(* CODESYS project Tc Motion Control.library
   Version: 0.1.0.0
   Title: Motion
   Author: Adam Garner
   Placeholder: Motion
   Company: Ljmu

Project tree, tasks and I/O mapping:
  libraries: Tc2_MC2, * (Beckhoff Automation GmbH); Tc2_MC2_Drive, * (Beckhoff Automation GmbH); Tc2_Standard, * (Beckhoff Automation GmbH); Tc2_System, * (Beckhoff Automation GmbH); Tc2_Utilities, * (Beckhoff Automation GmbH); Tc3_EventLogger, * (Beckhoff Automation GmbH); Tc3_JsonXml, * (Beckhoff Automation GmbH); Tc3_Module, * (Beckhoff Automation GmbH)
  DUTs/
    data type e_IDXBrakeState
    data type e_IDXError
    data type e_MCState
    data type e_MotorReadState
    data type ST_IDXError
    data type ST_IDXErrorCode
    data type ST_MCState
  GVLs/
  POUs/
    function block FB_IDXError [ST]: FB_init, GetErrorStructure, IsError, ResetError
    function block FB_IDXReadErrorCode [ST]: ParseErrorCode
    function block FB_IDXReadErrorRegister [ST]: ParseErrorRegister
    function block FB_IDXResetError [ST]: FB_init
    function block FB_Motion [ST]: Enable, Estop, FB_init, GetAxisRef, GetCurrentPosition, GetStatus, Home, MoveTo, Reset
    function block FB_MotionEventSender [ST]: COEError, EnableMotor, Homing, MotorError, MotorReset, MoveTo, NCError, NCReset
    function block FB_MotorBrake [ST]: Brake, BrakeStatus, EnableMotor, FB_init, UnitTestInputs
    function block FB_ReadErrorStringFromESI [ST]: FB_init, GetErrorString, StringToUint
    program MAIN [ST]
  VISUs/
*)

// DUTs/e_IDXBrakeState
{attribute 'qualified_only'}
{attribute 'strict'}
TYPE e_IDXBrakeState :
(
	Unpowered := 0,// no air in system brake on 
	Disengaging := 1, // Brake coming off 
	Disengaged :=2,// held off with compressed air
	Engaging	:=3, // brake coming online under command
	Engaged	:= 4,// brake on air in system 
	SafetyOverriden := 5, // safety override on brake on 
	SafetyActivating := 6, // safety override on brake Activing
	Unknown := 7,
	Error := 8
);
END_TYPE

// DUTs/e_IDXError
{attribute 'qualified_only'}
{attribute 'strict'}
TYPE e_IDXError :
(
	Generic_Error := 0,
	Current_Error :=1,
	Voltage_Error:=2,
	Temperature_Error:=3,
	Communication_Error := 4,
	Device_Profile_Specific := 5,
	Reserved := 6,
	Motion_Error :=7
);
END_TYPE

// DUTs/e_MCState
{attribute 'qualified_only'}
{attribute 'strict'}
TYPE e_MCState :
(
	Busy,
	Done,
	Error,
	CommandAborted,
	Active,
	Idle
);
END_TYPE

// DUTs/e_MotorReadState
// -27 as is qualified only shouldnt be flagged anyway
{attribute 'strict'}
{attribute 'qualified_only'}
TYPE e_MotorReadState :
(
Idle,
ReadingErrorArray,
{attribute 'analysis' := '-27'}
Parse,
EraseErrorArray,
Waiting,
Error,
CountingErrors,
ReadNextError

);
END_TYPE

// DUTs/ST_IDXError
TYPE ST_IDXError :
STRUCT
	GenericError:BOOL;
	CurrentError : BOOL;
	VoltageError:BOOL;
	TemperatureError:BOOL;
	Communication_Error :BOOL;
	DeviceProfileSpecific :BOOL;
	Reserved :BOOL;
	MotionError :BOOL;
	ErrorCodeArr:ARRAY [0..4] OF ST_IDXErrorCode;


END_STRUCT
END_TYPE

// DUTs/ST_IDXErrorCode
TYPE ST_IDXErrorCode :
STRUCT
	ErrorCode: UINT;
	ErrorString:STRING;
	TimeCode:DT;
END_STRUCT
END_TYPE

// DUTs/ST_MCState
TYPE ST_MCState :
STRUCT
	MCState : e_MCState;
	Done:BOOL;
	CommandAborted:BOOL;
	Status :BOOL;
	Active :BOOL;
	Busy:BOOL;
	Error:BOOL;
	ErrorID:UDINT;
	
END_STRUCT
END_TYPE

// POUs/FB_IDXError
FUNCTION_BLOCK FB_IDXError
// www.maxongroup.com/medias/sys_master/root/8837359632414/IDX-Firmware-Specification-En.pdf 	
VAR
	AxisName 				:STRING;
	ExecuteRead 			: BOOL; 
	MappedErrorCode AT%I* 	: UINT;
	stIDXError 				: ST_IDXError;
	
	fbIDXErrorEventSender 	: FB_MotionEventSender;
	MotorErrorEventSent		: BOOL;


	fbIdxReadErrorCode 		: FB_IDXReadErrorCode;
	NumOfErrorCodes			: USINT;
	ErrorCodeReadError 		: BOOL;
	ErrorCodeAdsErrorCode	: UINT;
	ErrorCodeReadBusy		: BOOL;
	
	fbIDXReadErrorRegister	: FB_IDXReadErrorRegister;
	ErrorRegisterReadError 	: BOOL;
	ErrorRegisterReadBusy	: BOOL;
	ErrorRegisterAdsErrorCode: UINT;
	
	fbReadErrorStringFromESI: FB_ReadErrorStringFromESI(FileNameIn := 'C:\ProgramData\Beckhoff\TwinCAT\3.1\Repository\Beckhoff Automation GmbH\maxon_motor_IDX_0170h_6650h_0000h_0000h_ESI.xml');
	ErrorStringReadReady 	: BOOL;
	ErrorStringReadBusy 	: BOOL;
	ErrorStringReadError 	: BOOL;
	ErrorStringFound 		: BOOL;
	
	CoeErrorCodeMessageSent : BOOL;
	CoeErrorregisterMessageSent : BOOL;
	
	

	

END_VAR

VAR_INPUT
	Axis 					: AXIS_REF;
END_VAR

VAR_OUTPUT
    Busy         			: BOOL;
    Error        			: BOOL;
END_VAR

VAR CONSTANT
	MaxIndex 				: USINT := 4;
END_VAR

VAR_TEMP
	TempErrorCode 			: UINT;
	TempErrorString 		: STRING;
	Index					: USINT;
END_VAR

// read error Reg 
// check for error messages availible 

IF NOT (MappedErrorCode=0) THEN
	ExecuteRead := TRUE; // motor in error state 
	
ELSE
	ExecuteRead:= FALSE;
END_IF

fbIdxReadErrorCode(
	Axis:= Axis,
	Execute:= ExecuteRead,
	NumOfErrors=> NumOfErrorCodes,
	stErrorInOut:=stIDXError,
	ReadError=>ErrorCodeReadError,
	AdsErrId=>ErrorCodeAdsErrorCode,
	ReadBusy => ErrorCodeReadBusy);

CoeErrorCodeMessageSent := fbIDXErrorEventSender.COEError(
	AxisName := AxisName,
	Error := ErrorCodeReadError,
	AdsErrId:= ErrorCodeAdsErrorCode,
	Description:= 'ErrorCodeRead');

fbIDXReadErrorRegister(
	Axis:= Axis, 
	Execute:= ExecuteRead, 
	stErrorRegisterInOut:=stIDXError , 
	ReadError=> ErrorRegisterReadError, 
	AdsErrId=> ErrorRegisterAdsErrorCode, 
	ReadBusy=> ErrorRegisterReadBusy );

CoeErrorregisterMessageSent:= fbIDXErrorEventSender.COEError(
	AxisName:= AxisName,
	Error := ErrorRegisterReadError,
	AdsErrId:= ErrorRegisterAdsErrorCode,
	Description:= 'ErrorCodeRegister');


fbReadErrorStringFromESI(
	ReadyFlag=>ErrorStringReadReady,
	Busy=>ErrorStringReadBusy,
	Error=>ErrorStringReadError);


IF (ErrorStringReadReady AND ExecuteRead ) THEN
	FOR Index:=0  TO MaxIndex BY 1 DO
		TempErrorCode:= stIDXError.ErrorCodeArr[Index].ErrorCode;
		IF NOT (TempErrorCode =0) THEN
			ErrorStringFound:= fbReadErrorStringFromESI.GetErrorString(ErrorCodeIn:= TempErrorCode,ErrorStringOut=>TempErrorString);
			stIDXError.ErrorCodeArr[Index].ErrorString:= TempErrorString;
		END_IF
	END_FOR
END_IF
	
MotorErrorEventSent:= fbIDXErrorEventSender.MotorError(stIDXError:=stIDXError,AxisName:= AxisName);

Busy := ErrorStringReadBusy OR ErrorRegisterReadBusy OR ErrorCodeReadBusy;
Error := ErrorStringReadError OR ErrorRegisterReadError OR ErrorCodeReadError;

METHOD FB_init : BOOL
VAR_INPUT
	bInitRetains : BOOL; // if TRUE, the retain variables are initialized (warm start / cold start)
	bInCopyCode : BOOL;  // if TRUE, the instance afterwards gets moved into the copy code (online change)
	AxisNameIn	:String;
END_VAR
AxisName := AxisNameIn;
END_METHOD

METHOD PUBLIC GetErrorStructure 
VAR_OUTPUT
	StIDXErrorOut : ST_IDXError;
END_VAR
StIDXErrorOut:= stIDXError;
END_METHOD

// returns true if motor is in error state 
METHOD IsError : BOOL
IsError := ExecuteRead;
END_METHOD

METHOD ResetError : BOOL
VAR_IN_OUT
	   		{attribute 'analysis' := '-27'}
	Execute			: BOOL;(*Function block execution is triggered by a rising edge at this input.*)
END_VAR

VAR_INST
	fbCoEWrite		: FB_CoEWrite;
    Data       		: UINT := 16#0080;
    ReadError          	: BOOL;
    AdsErrId       	: UINT;
    CANopenErrId   	: UINT;
END_VAR

VAR CONSTANT
	NetId          	: T_AmsNetID:= '';(*netID of PC with NC*)
   	Index          	: WORD:= 16#6040;(*CoE object index*)
   	SubIndex       	: BYTE:=16#0;(*CoE sub index*)
   	Timeout        	: TIME := DEFAULT_ADS_TIMEOUT;(*States the time before the function is cancelled.*)
  	CompleteAccess 	: BOOL:= FALSE;(*Function block reads the complete object with all sub index*)
END_VAR
IF __ISVALIDREF(Execute) THEN	
	fbCoEWrite(
    NetId          := NetId, 
    Index          := Index, 
    SubIndex       := SubIndex, 
    pSrcBuf        := ADR(Data), 
    BufLen         := USINT_TO_UDINT(SIZEOF(Data)), 
    Execute        := Execute, 
    Timeout        := Timeout, 
    CompleteAccess := CompleteAccess, 
    Axis := Axis
);

END_IF

IF (NOT fbCoEWrite.Busy) AND   __ISVALIDREF(Execute) THEN
    ReadError    := fbCoEWrite.Error;
	IF (NOT ReadError) AND Execute THEN
		ResetError:= TRUE; // reset successfully only shows for one cycle
	ELSE 
		ResetError:= FALSE;
	END_IF
	
    AdsErrId     := fbCoEWrite.AdsErrId;
    CANopenErrId :=fbCoEWrite.CANopenErrId;
    Execute      := FALSE;
	IF NOT ReadError THEN
		ResetError:= TRUE; // reset successfully
	END_IF
END_IF
END_METHOD

END_FUNCTION_BLOCK

// POUs/FB_MotionEventSender
{attribute 'analysis' := '-2'} // empty function block
// this fb is used to generate events via methods used in this libary 
FUNCTION_BLOCK INTERNAL FB_MotionEventSender
VAR
	fbTcMessage : FB_TcMessage;
END_VAR

// returns true for one cycle when event is generated 
// method is used for events in a Coe read/write 
METHOD INTERNAL COEError : BOOL

VAR_INPUT
    Error        	: BOOL; // from COE read/write 
    AdsErrId     	: UINT; // from COE read/write 
	Description		: STRING; // description of what the COE was doing eg MotorError Read or MotorReset Write is displayed in event
	AxisName		:STRING; // for display in event 
END_VAR
VAR_INST //previous cycle results
	LastError		:BOOL; 

END_VAR

VAR
	SendResult 			:HRESULT;

END_VAR
COEError := FALSE;
IF (NOT LastError) AND Error THEN // only enter is a current error is in place and the last cycle the error was 0 
	 {analysis -9,-46} // Unused  return values and possible use of none init interfaces 
	fbTcMessage.CreateEx(TC_EVENTS.MotionEvents.CoeError,0);
	fbTcMessage.ipArguments.Clear();
	fbTcMessage.ipArguments.AddString(AxisName);
	fbTcMessage.ipArguments.AddUInt(AdsErrId);
	fbTcMessage.ipArguments.AddString(Description);
	SendResult:= fbTcMessage.Send(0);
	{analysis 9,46}
	IF (SendResult=0) THEN
		COEError := TRUE;
	END_IF
END_IF
LastError:= Error;
END_METHOD

// method generates events when axis is enabled / disabled 
// returns true for one cycle when event is generated 
METHOD INTERNAL EnableMotor 		: BOOL
VAR_IN_OUT
	stAxisPowerState 	: ST_MCState; //structure from fb motion libary shows movement FB status 
END_VAR
VAR_INPUT
	AxisName 			:STRING; // displayed in event 
END_VAR
VAR_INST //previous cycle results
	stLastAxisPowerState :ST_MCState;
END_VAR
VAR
	SendResult 			: HRESULT;
	SendEvent 			: BOOL := FALSE;
END_VAR
EnableMotor := FALSE;

IF __ISVALIDREF(stAxisPowerState) THEN

	IF NOT (stLastAxisPowerState.MCState = stAxisPowerState.MCState) THEN // state has changed 
	 	{analysis -9,-46} // Unused  return values and possible use of none init interfaces 
		CASE(stAxisPowerState.MCState) OF
		
		e_MCState.Active:
			fbTcMessage.CreateEx(TC_EVENTS.MotionEvents.MotorEnabled,0);
			SendEvent:= TRUE;
		
		e_MCState.Error:
			fbTcMessage.CreateEx(TC_EVENTS.MotionEvents.MotorEnableError,0);
			SendEvent:= TRUE;
		
		e_MCState.Idle:
			fbTcMessage.CreateEx(TC_EVENTS.MotionEvents.MotorDisabled,0);
			SendEvent:= TRUE;
		ELSE
			SendEvent:= FALSE;
		END_CASE
	
		IF SendEvent THEN
			fbTcMessage.ipArguments.Clear();
			fbTcMessage.ipArguments.AddString(AxisName);
			SendResult:= fbTcMessage.Send(0);
			IF (SendResult=0) THEN
				EnableMotor := TRUE;
			END_IF
		END_IF
	END_IF

	stLastAxisPowerState := stAxisPowerState;
END_IF
END_METHOD

// returns true for one cycle when event is generated 
// creates events during homing
// returns true for one cycle when event is generated 
METHOD INTERNAL Homing : BOOL
VAR_IN_OUT
	stAxisHomeState : ST_MCState; //structure from fb motion libary shows movement FB status 
END_VAR
VAR_INPUT
	AxisName :STRING; // displayed in event 
 
END_VAR
VAR_INST //previous cycle results
	stLastAxisHomeState : ST_MCState;
END_VAR
VAR
	SendEvent : BOOL;
	SendResult : Hresult;
END_VAR
Homing := FALSE;

IF  __ISVALIDREF(stAxisHomeState) THEN
	
	IF  (NOT (stLastAxisHomeState.MCState = stAxisHomeState.MCState)) THEN
		CASE(stAxisHomeState.MCState) OF 
		{analysis -9,-46} // Unused  return values and possible use of none init interfaces 
		e_MCState.Done:
			fbTcMessage.CreateEx(TC_EVENTS.MotionEvents.HomeCompleted,0);
			fbTcMessage.ipArguments.Clear();
			fbTcMessage.ipArguments.AddString(AxisName);
			SendEvent := TRUE;
		
		e_MCState.Busy:
			fbTcMessage.CreateEx(TC_EVENTS.MotionEvents.HomeCommandReceived,0);
			fbTcMessage.ipArguments.Clear();
			fbTcMessage.ipArguments.AddString(AxisName);
			SendEvent := TRUE;
		
		e_MCState.Error:
			fbTcMessage.CreateEx(TC_EVENTS.MotionEvents.HomeError,0);
			fbTcMessage.ipArguments.Clear();
			fbTcMessage.ipArguments.AddString(AxisName);
			fbTcMessage.ipArguments.AddUDInt(stAxisHomeState.ErrorID);
			SendEvent := TRUE;
			
		
		e_MCState.CommandAborted:
			fbTcMessage.CreateEx(TC_EVENTS.MotionEvents.HomeAborted,0);
			fbTcMessage.ipArguments.Clear();
			fbTcMessage.ipArguments.AddString(AxisName);
			SendEvent := TRUE;
			
		e_MCState.Idle:
			SendEvent := FALSE;
		
		ELSE
			SendEvent := FALSE;
			
		
		END_CASE
		
			IF SendEvent THEN
				SendResult:= fbTcMessage.Send(0);
			
				IF (SendResult=0) THEN
					Homing := TRUE;
				END_IF
	
			END_IF
	END_IF
	
	stLastAxisHomeState:= stAxisHomeState;

END_IF
END_METHOD

// genereates events about a motor controllers errors it loops through the array of data errors in St_IDXError
// returns true for one cycle when event is generated 
METHOD INTERNAL MotorError :BOOL
VAR_IN_OUT
	stIDXError 	:ST_IDXError;
END_VAR
VAR_INPUT
	AxisName 	:STRING;  // displayed in event 
END_VAR
VAR_INST //previous cycle results
	stLastIDXError : ST_IDXError;
END_VAR
VAR
	Index :INT;
	ErrorCodeInHex :STRING[255];
	SendResult :HRESULT;
END_VAR
VAR CONSTANT
	MaxIndex :INT := 4 ; // upper limit of loop 
END_VAR
MotorError:= FALSE;
IF __ISVALIDREF(stIDXError) THEN
FOR Index := 0 TO MaxIndex BY 1 DO 
	IF NOT ( stIDXError.ErrorCodeArr[Index].ErrorCode =stLastIDXError.ErrorCodeArr[Index].ErrorCode) THEN
		{analysis -9,-46,-130}// Unused  return values possible use of none init interfaces ,  Implicit expanding conversion 
		fbTcMessage.CreateEx(TC_EVENTS.MotionEvents.MotorError,0);
		fbTcMessage.ipArguments.Clear();
		fbTcMessage.ipArguments.AddString(AxisName);
		ErrorCodeInHex := DWORD_TO_HEXSTR(stIDXError.ErrorCodeArr[Index].ErrorCode,4,FALSE); // error code as hex string 
		fbTcMessage.ipArguments.AddString(ErrorCodeInHex);
		fbTcMessage.ipArguments.AddString(stIDXError.ErrorCodeArr[Index].ErrorString);
		SendResult := fbTcMessage.Send(0);
		{analysis 9,46,130}
		IF (SendResult=0) THEN
			MotorError:= TRUE;
		END_IF
		stLastIDXError.ErrorCodeArr[Index]:= stIDXError.ErrorCodeArr[Index];
			
	END_IF
END_FOR
END_IF
END_METHOD

// events for resetting a motor controller 
// returns true for one cycle when event is generated 
METHOD INTERNAL MotorReset : BOOL
VAR_IN_OUT
	stAxisResetState : ST_MCState;
END_VAR
VAR_INPUT
	AxisName :STRING; // displayed in event
	ErrorCodeIn :UDINT;
END_VAR
VAR_INST//previous cycle results
	stLastAxisResetState : ST_MCState;
END_VAR
VAR
	SendEvent : BOOL;
	SendResult : Hresult;
END_VAR
MotorReset := FALSE;

IF  __ISVALIDREF(stAxisResetState) THEN
	
	IF  (NOT (stLastAxisResetState.MCState = stAxisResetState.MCState)) THEN
		CASE(stAxisResetState.MCState) OF 
		{analysis -9,-46} // Unused  return values and possible use of none init interfaces 
		e_MCState.Done:
			fbTcMessage.CreateEx(TC_EVENTS.MotionEvents.MotorResetCompleted,0);
			fbTcMessage.ipArguments.Clear();
			fbTcMessage.ipArguments.AddString(AxisName);
			SendEvent := TRUE;
		
		e_MCState.Busy:
			fbTcMessage.CreateEx(TC_EVENTS.MotionEvents.MotorResetReceived,0);
			fbTcMessage.ipArguments.Clear();
			fbTcMessage.ipArguments.AddString(AxisName);
			SendEvent := TRUE;
		
		e_MCState.Error:
			SendEvent := FALSE;
			
		e_MCState.Idle:
			SendEvent := FALSE;
		
		ELSE
			SendEvent := FALSE;
			
		
		END_CASE
		
			IF SendEvent THEN
				SendResult:= fbTcMessage.Send(0);
			
				IF (SendResult=0) THEN
					MotorReset := TRUE;
				END_IF
	
			END_IF
	END_IF
	
	stLastAxisResetState:= stAxisResetState;

END_IF
END_METHOD

// method used to generate events on movement commands 
// moveTo bool is true when a event has been sent 
METHOD MoveTo : BOOL
VAR_IN_OUT
	stAxisMoveState : ST_MCState;
END_VAR
VAR_INPUT
	AxisName :STRING;// displayed in event
	TargetPositionIn : LREAL;
	VelocityIn : LREAL;
END_VAR
VAR_INST//previous cycle results
	stLastAxisMoveState : ST_MCState;
END_VAR
VAR
	SendEvent : BOOL;
	SendResult : Hresult;
	
END_VAR
MoveTo:= FALSE;
	
IF __ISVALIDREF(stAxisMoveState) THEN
	
	IF  (NOT (stAxisMoveState.MCState = stLastAxisMoveState.MCState)) THEN
	
		CASE(stAxisMoveState.MCState) OF 
		{analysis -9,-46} // Unused  return values and possible use of none init interfaces 	
			e_MCState.Active:
			fbTcMessage.CreateEx(TC_EVENTS.MotionEvents.MotorMoveActive,0);
			fbTcMessage.ipArguments.Clear();
			fbTcMessage.ipArguments.AddString(AxisName);
			SendEvent := TRUE;
	
		e_MCState.Busy:
			fbTcMessage.CreateEx(TC_EVENTS.MotionEvents.MoveCommandReceived,0);
			fbTcMessage.ipArguments.Clear();
			fbTcMessage.ipArguments.AddString(AxisName);
			fbTcMessage.ipArguments.AddLReal(TargetPositionIn);
			fbTcMessage.ipArguments.AddLReal(VelocityIn);
			SendEvent := TRUE;
	
		e_MCState.Error:
			fbTcMessage.CreateEx(TC_EVENTS.MotionEvents.MotorMoveError,0);
			fbTcMessage.ipArguments.Clear();
			fbTcMessage.ipArguments.AddString(AxisName);
			fbTcMessage.ipArguments.AddUDInt(stAxisMoveState.ErrorID);
			SendEvent := TRUE;
	
		e_MCState.CommandAborted:
			fbTcMessage.CreateEx(TC_EVENTS.MotionEvents.MovementAborted,0);
			fbTcMessage.ipArguments.Clear();
			fbTcMessage.ipArguments.AddString(AxisName);
			SendEvent := TRUE;
	
		e_MCState.Done:
			fbTcMessage.CreateEx(TC_EVENTS.MotionEvents.MotorMoveFinshed,0);
			fbTcMessage.ipArguments.Clear();
			fbTcMessage.ipArguments.AddString(AxisName);
			fbTcMessage.ipArguments.AddLReal(TargetPositionIn);
			SendEvent := TRUE;
	
		e_MCState.Idle:
			SendEvent := FALSE;
	
	
		ELSE
			SendEvent := FALSE;
		
		END_CASE
		
		IF SendEvent THEN
			SendResult:= fbTcMessage.Send(0);
			
			IF (SendResult=0) THEN
				MoveTo := TRUE;
			END_IF
		
		END_IF
	
		stLastAxisMoveState := stAxisMoveState;
	
	END_IF

END_IF
END_METHOD

// method creates events for NC block Errors 
// returns true for one cycle when event is generated 
METHOD INTERNAL NCError : BOOL
VAR_IN_OUT
	stAxisStatus : ST_AxisStatus;
END_VAR
VAR_INPUT
	AxisName 	:STRING; // displayed in event
END_VAR
VAR_INST//previous cycle results
	stLastAxisErrorID :UDINT;
END_VAR
VAR
	SendResult :HRESULT;
END_VAR
NCError:= FALSE;
IF __ISVALIDREF(stAxisStatus) THEN

	IF NOT ( stAxisStatus.ErrorID = stLastAxisErrorID) THEN
		{analysis -9,-46,-130}// Unused  return values possible use of none init interfaces ,  Implicit expanding conversion 
		fbTcMessage.CreateEx(TC_EVENTS.MotionEvents.NCError,0);
		fbTcMessage.ipArguments.Clear();
		fbTcMessage.ipArguments.AddString(AxisName);
		fbTcMessage.ipArguments.AddUDInt(stAxisStatus.ErrorID);
		SendResult := fbTcMessage.Send(0);
		{analysis 9,46,130}
		IF (SendResult=0) THEN
			NCError:= TRUE;
		END_IF
		stLastAxisErrorID:= stAxisStatus.ErrorID;
			
	END_IF
END_IF
END_METHOD

// creates events during a NCreset 
// returns true for one cycle when event is generated 
METHOD INTERNAL NCReset : BOOL
VAR_IN_OUT
	stAxisResetState : ST_MCState;
	
END_VAR
VAR_INPUT
	AxisName :STRING;// displayed in event
	ErrorCodeIn :UDINT;
END_VAR
VAR_INST//previous cycle results
	stLastAxisResetState : ST_MCState;
END_VAR
VAR
	SendEvent : BOOL;
	SendResult : Hresult;
END_VAR
NCReset := FALSE;

IF  __ISVALIDREF(stAxisResetState) THEN
	
	IF  (NOT (stLastAxisResetState.MCState = stAxisResetState.MCState)) THEN
		CASE(stAxisResetState.MCState) OF 
		{analysis -9,-46} // Unused  return values and possible use of none init interfaces 
		e_MCState.Done:
			fbTcMessage.CreateEx(TC_EVENTS.MotionEvents.NCResetCompleted,0);
			fbTcMessage.ipArguments.Clear();
			fbTcMessage.ipArguments.AddString(AxisName);
			SendEvent := TRUE;
		
		e_MCState.Busy:
			fbTcMessage.CreateEx(TC_EVENTS.MotionEvents.NCResetReceived,0);
			fbTcMessage.ipArguments.Clear();
			fbTcMessage.ipArguments.AddString(AxisName);
			SendEvent := TRUE;
		
		e_MCState.Error:
			fbTcMessage.CreateEx(TC_EVENTS.MotionEvents.NCResetError,0);
			fbTcMessage.ipArguments.Clear();
			fbTcMessage.ipArguments.AddString(AxisName);
			fbTcMessage.ipArguments.AddUDInt(ErrorCodeIn);
			SendEvent := TRUE;
			
		e_MCState.Idle:
			SendEvent := FALSE;
		
		ELSE
			SendEvent := FALSE;
			
		
		END_CASE
		
			IF SendEvent THEN
				SendResult:= fbTcMessage.Send(0);
			
				IF (SendResult=0) THEN
					NCReset := TRUE;
				END_IF
	
			END_IF
	END_IF
	
	stLastAxisResetState:= stAxisResetState;

END_IF
END_METHOD

END_FUNCTION_BLOCK

// POUs/FB_IDXReadErrorCode
// function to read the Diagnosis history odject of a IDX motor 
// this fb will read the errors in the error array looping between them with a 1s pause between reads
// if execute is false it resets the error array no none 
// www.maxongroup.com/medias/sys_master/root/8837359632414/IDX-Firmware-Specification-En.pdf
// definition of motor structure on 6.2.12 pg 71

FUNCTION_BLOCK FB_IDXReadErrorCode
VAR CONSTANT
	 NetId             : T_AmsNetID := ''; // assumes local machine 
    Index             : WORD := 16#10F3; // diagnosis history 
    Timeout           : TIME := T#5S;
    CompleteAccess    : BOOL := FALSE; // to read the whole index in one go instead of sunindexs
	NumberOfErrors :USINT := 5; // number of errors 
	MaxErrorIndex :USINT := 4; // max index so one below number of errors 
	MotorErrorSubindexStart :USINT := 6 ;
END_VAR
VAR_INPUT
	Axis :AXIS_REF;// used For Coe read 
		 {attribute 'analysis' := '-27'}
	Execute: BOOL;	
END_VAR
VAR_IN_OUT
	stErrorInOut : ST_IDXError;// a array for errors with code string and datetime 
END_VAR
VAR_OUTPUT
	NumOfErrors :USINT; // how man errors are present 
	ReadError :BOOL; // error reading motor 
	AdsErrId  : UINT; //holds Reading error codes 
	ReadBusy:BOOL;
END_VAR

VAR
	eMotorReadState : e_MotorReadState; // enum of fb  current state
	
	CoETimer : TON:= (PT:= T#1S); // timer 
	TimerStart:BOOL:= FALSE;
	TimerElapsed:BOOL;
	fbCoERead         : FB_CoERead; // fb to Coe read
    SubIndex          : BYTE := 16#6;  // first error index 
    ExecuteRead       : BOOL := FALSE;
    Error             : BOOL;
    CANopenErrId      : UINT; 
	ParsingError	: BOOL;
	
	ParsedErrorCode : ST_IDXErrorCode;
	ErrorIndex :BYTE := 0; // where to save the error code in the error array 
	RawErrorArray :ARRAY[0..15] OF USINT; // buffer to store the raw CoE Read
	EmptyError : ST_IDXError; // used to reinitalise the error array while not in error state 
END_VAR
VAR_TEMP
		ArrayIndex:USINT;
END_VAR


fbCoERead(
    NetId          := NetId, 
    Index          := Index, 
    SubIndex       := SubIndex, 
    pDstBuf        := ADR(RawErrorArray), 
    BufLen         := SIZEOF(RawErrorArray), 
    Execute        := ExecuteRead, 
    Timeout        := Timeout, 
    CompleteAccess := CompleteAccess, 
    Axis           := Axis,
	Busy			=> ReadBusy 
); // read the Coe 



CoETimer(IN:= TimerStart,Q=>TimerElapsed); // process timer

CASE(eMotorReadState) OF 
	
e_MotorReadState.Idle: // not reading
	//reset counters
	SubIndex := MotorErrorSubindexStart ;// first error in  motor error array
	ErrorIndex := 0; // first error in output array
	NumOfErrors:= 0;
	
	IF Execute THEN
		ExecuteRead := TRUE;
		eMotorReadState := e_MotorReadState.ReadingErrorArray;
	ELSE 
		IF __ISVALIDREF(stErrorInOut) THEN
			stErrorInOut:= EmptyError; 
		 END_IF
	END_IF

e_MotorReadState.ReadingErrorArray:

IF NOT (fbCoERead.Busy) THEN // finished reading so write any errors to varibles 
	Error        :=fbCoERead.Error; 
    AdsErrId     :=fbCoERead.AdsErrId;
    CANopenErrId :=fbCoERead.CANopenErrId;
    ExecuteRead  := FALSE; // Reset Reading FB
    
	ReadError:= Error; // if a read fails put into error state 
	ParseErrorCode(ErrorArrayIn:= RawErrorArray,ParsedErrorOut=> ParsedErrorCode,Error=> ParsingError);
	
	IF NOT ParsingError OR Error THEN // if errored dont write to array 
	stErrorInOut.ErrorCodeArr[ErrorIndex]:= ParsedErrorCode;
	END_IF
	
	IF (ErrorIndex = MaxErrorIndex) THEN //  has read whole array 
		eMotorReadState := e_MotorReadState.CountingErrors; //Count and then waiting timer on next cycle
	ELSE
		eMotorReadState:= e_MotorReadState.ReadNextError;
	END_IF
	

	
	
END_IF

e_MotorReadState.ReadNextError:

ErrorIndex := (ErrorIndex+1) MOD NumberOfErrors; // loop from the error indexs 0 to 4 
SubIndex := ErrorIndex + MotorErrorSubindexStart; // IDX Subindex to read from the motor subindexs 6 to 10 contain errors 
ExecuteRead:= TRUE;
eMotorReadState:= e_MotorReadState.ReadingErrorArray;

e_MotorReadState.CountingErrors:
NumOfErrors := 0;
IF __ISVALIDREF(stErrorInOut) THEN
	FOR ArrayIndex := 0 TO MaxErrorIndex BY 1 DO 
		IF NOT (stErrorInOut.ErrorCodeArr[ArrayIndex].ErrorCode =0) THEN 
		 {analysis -38}
			NumOfErrors := (NumOfErrors +1);
		END_IF
	END_FOR
END_IF
eMotorReadState := e_MotorReadState.Waiting;

e_MotorReadState.Waiting:
TimerStart:= TRUE; // start waiting timer 
IF TimerElapsed THEN
	TimerStart:= FALSE; // reset timer 
	eMotorReadState := e_MotorReadState.Idle; // back to begining 
END_IF

e_MotorReadState.Parse:
// no code needed
e_MotorReadState.EraseErrorArray:
// no code needed

e_MotorReadState.Error:
SubIndex := 6 ;// first error in  motor error array
ErrorIndex := 0; // first error in output array
// Erase error array as not currently reading error 
NumOfErrors:= 0;
ExecuteRead := FALSE;
eMotorReadState := e_MotorReadState.Idle;		



ELSE 
	eMotorReadState := e_MotorReadState.Idle;

END_CASE



// example packet for error 8A81
//00 E0 81 8A 02 00 81 8A 00 00 00 00 00 00 00 00
//0  1  2  3  4  5  6  7  8  9  10 11 12 13 14 15

METHOD ParseErrorCode  
VAR_IN_OUT
ErrorArrayIn :ARRAY[0..15] OF USINT;
END_VAR

VAR_OUTPUT
	ParsedErrorOut : ST_IDXErrorCode;
	Error:BOOL;
END_VAR

VAR
	RawErrorCodes : ARRAY [0..1] OF UINT;
	FirstErrorByte : UINT;
	SecondErrorByte : UINT;
	
END_VAR

VAR CONSTANT
	BlankArray : ARRAY[0..15] OF USINT := [0,0,0,0,0,0,0,0,0,0,0,0,0,0,0,0] ;
END_VAR
Error:= FALSE;
IF __ISVALIDREF(ErrorArrayIn) THEN
	// grab from the first time the error is wrote packets 3&4
	FirstErrorByte := SHL(USINT_TO_UINT(ErrorArrayIn[3]),8);// grab first byte and shift left 
	SecondErrorByte := USINT_TO_UINT(ErrorArrayIn[2]);  // grab second byte 
	RawErrorCodes[0] := FirstErrorByte OR SecondErrorByte; // combine 

	// grab from the Second time the error is wrote packets 6&7
	FirstErrorByte := SHL(USINT_TO_UINT(ErrorArrayIn[7]),8);// grab first byte and shift left 
	SecondErrorByte := USINT_TO_UINT(ErrorArrayIn[6]);  // grab second byte 
	RawErrorCodes[1] := FirstErrorByte OR SecondErrorByte; // combine 
ELSE 
	Error:= TRUE;
END_IF

IF NOT RawErrorCodes[0] = RawErrorCodes[1] THEN
	Error:= TRUE;
ELSE
	ParsedErrorOut.ErrorCode:= RawErrorCodes[0]; 

	


END_IF
// clear array after parsing 
ErrorArrayIn := BlankArray;
END_METHOD

END_FUNCTION_BLOCK

// POUs/FB_IDXReadErrorRegister
FUNCTION_BLOCK FB_IDXReadErrorRegister
VAR_INPUT
	Axis :AXIS_REF;// used For Coe read 
	Execute: BOOL;	
END_VAR
VAR_IN_OUT
	stErrorRegisterInOut :  ST_IDXError;// a array for errors with code string and datetime 
END_VAR
VAR_OUTPUT
	ReadError :BOOL; // error reading motor 
	AdsErrId  : UINT; //holds Reading error codes 
	ReadBusy :BOOL;
END_VAR

VAR
	
	eMotorReadState : e_MotorReadState; // enum of fb  current state
	CoETimer : TON:= (PT:= T#1S); // timer 
	TimerStart:BOOL:= FALSE;
	TimerElapsed:BOOL;
	fbCoERead         : FB_CoERead; // fb to Coe read
    ExecuteRead       : BOOL := FALSE;
    Error             : BOOL;
	Busy				:BOOL;
    CANopenErrId      : UINT;
	RawErrorRegister : USINT; // buffer to store the raw CoE Read
	EmptyError : ST_IDXError; // used to reinitalise the error array while not in error state
END_VAR
VAR CONSTANT
	NetId             : T_AmsNetID := ''; // assumes local machine 
    Index             : WORD := 16#1001; // diagnosis history 
    SubIndex          : BYTE := 16#0;  // first error index
	Timeout           : TIME := T#5S;
    CompleteAccess    : BOOL := FALSE; // to read the whole index in one go instead of sunindexs
	
END_VAR

{analysis -130} // widening conversion fine in this context  of buflen
fbCoERead(
    NetId          := NetId, 
    Index          := Index, 
    SubIndex       := SubIndex, 
    pDstBuf        := ADR(RawErrorRegister),
    BufLen         := SIZEOF(RawErrorRegister), 
    Execute        := ExecuteRead, 
    Timeout        := Timeout, 
    CompleteAccess := CompleteAccess, 
    Axis           := Axis,
	Busy			=> Busy 
); // read the Coe 
{analysis +130}
ReadBusy := Busy;


CoETimer(IN:= TimerStart,Q=>TimerElapsed); // process timer

CASE(eMotorReadState) OF 
	
e_MotorReadState.Idle: // not reading
	IF Execute THEN
	ExecuteRead := TRUE;
	eMotorReadState := e_MotorReadState.ReadingErrorArray;
	ELSE // Erase error array as not currently reading error 
		IF __ISVALIDREF(stErrorRegisterInOut) THEN
			stErrorRegisterInOut:= EmptyError;
		END_IF
	END_IF

e_MotorReadState.ReadingErrorArray:
IF NOT Busy THEN // finished reading so write any errors to varibles 
	Error        :=fbCoERead.Error; 
    AdsErrId     :=fbCoERead.AdsErrId;
    CANopenErrId :=fbCoERead.CANopenErrId;
    ExecuteRead      := FALSE; // Reset Reading FB as finished reading
	ReadError:= Error; // if a read fails Flag Error
	IF NOT Error  THEN// add data to structure
		 {analysis -145} //not init ref , it is checked for valid reference inside function 
		ParseErrorRegister(ErrorRegIn:= RawErrorRegister,StErrorRegister:= stErrorRegisterInOut);
 		{analysis +145} 
	END_IF
	eMotorReadState := e_MotorReadState.Waiting; // start the waiting timer 
END_IF

e_MotorReadState.Waiting:
TimerStart:= TRUE; // start waiting timer 
IF TimerElapsed THEN
	TimerStart:= FALSE; // reset timer 
	eMotorReadState := e_MotorReadState.Idle; // back to begining 
END_IF
e_MotorReadState.Error:
IF NOT Execute THEN
	eMotorReadState := e_MotorReadState.Idle;
END_IF

ELSE
	eMotorReadState := e_MotorReadState.Error;
	
END_CASE

METHOD ParseErrorRegister 
VAR_INPUT
	ErrorRegIn :USINT;
END_VAR
VAR_IN_OUT
	StErrorRegister :ST_IDXError;
END_VAR
IF __ISVALIDREF(StErrorRegister) THEN	
	StErrorRegister.GenericError := ErrorRegIn.0;
	StErrorRegister.CurrentError := ErrorRegIn.1;
	StErrorRegister.VoltageError := ErrorRegIn.2;
 	StErrorRegister.TemperatureError := ErrorRegIn.3;
	StErrorRegister.Communication_Error := ErrorRegIn.4;
	StErrorRegister.DeviceProfileSpecific := ErrorRegIn.5;
	StErrorRegister.MotionError := ErrorRegIn.7;
END_IF
END_METHOD

END_FUNCTION_BLOCK

// POUs/FB_ReadErrorStringFromESI
// this FB reads the ESI file given in Fbinit navigates to the DiagMessages and takes the error strings and populates them into a error array for reading out 
// the code only adds 25 errors per cycle so can take many cycles to populate the whole array this is done once on bootup
// and has a ready flag indicating when its complete
// once populated the geterrorstring method is used to pull the error strings for displaying to user 

// the ESI structure is below except with more error codes 

//<EtherCATInfo Version="1.2" xmlns:xsi="http://www.w3.org/2001/XMLSchema-instance" xsi:noNamespaceSchemaLocation="EtherCATInfo.xsd">
// 	<Descriptions>
//		<Devices>
//			<Device Physics="YY">
//				<Profile>
//					<DiagMessages>
//						<DiagMessage>
//             				<TextId>#x0000</TextId>
//             				<MessageText>None</MessageText>
//           			</DiagMessage>
//           			<DiagMessage>
//            				<TextId>#x1000</TextId>
//            				<MessageText>Generic error</MessageText>
//          			</DiagMessage>
//					<DiagMessages>
//				</Profile>
//			</Device Physics="YY">
//		</Devices>
// 	</Descriptions>
//</EtherCATInfo Version="1.2" xmlns:xsi="http://www.w3.org/2001/XMLSchema-instance" xsi:noNamespaceSchemaLocation="EtherCATInfo.xsd">


FUNCTION_BLOCK FB_ReadErrorStringFromESI
VAR_OUTPUT
	Busy:BOOL; // is busy when reading and parsing file 
	Error :BOOL; 
	ReadyFlag :BOOL; // once error array is populated
END_VAR
VAR
	FileName :STRING[255]; // file path of ESI file to parse 
	{attribute 'strict'}
	eXMLReadState : (LoadingFile,GettingIterator,ParsingFile,Ready,ErrorState); // used in case switch statement
	ErrorCodeStringArray : ARRAY [0..16#FFFF] OF STRING;
	fbXml : FB_XmlDomParser; // init fbto parse the XML  
	LoadFile:BOOL:= TRUE; // used to trigger FBXMl to start reading  
	FileLoaded:BOOL; // latches true once file opened
	xmlDoc: SXmlNode; // root node
	xmlEtherCatInfo :SXmlNode; // <ethercatInfo> Node
	xmlDescriptions :SXmlNode;// <Descriptions> Node 
	xmlDevices : SXmlNode; // <Devices> Node 
	xmlDevice : SXmlNode;// <Device Physics="YY"> Node 
	xmlProfile : SXmlNode;//<Profile> Node
	xmlDiagMessages:SxmlNode;// <DiagMessages> Node
	xmlDiagmessageIterator:SXmlIterator;//<DiagMessage> iterator
	xmlDiagMessage :SXmlNode; // individual <DiagMessage> nodes
	xmlDiagMessageIDNode :sxmlNode; // individual <TextId> node
	xmlDiagMessageMessageTextNode : SxmlNode;// individual <MessageText> node
	xmlDiagMessageIDText:STRING[8];
	ErrorCode :UINT;
	StringToUintError :BOOL;
	

END_VAR
VAR CONSTANT
	NumToItetratePerCycle :UINT := 25; // controls number of messages read in a cycle 
END_VAR
VAR_TEMP
	
	ErrorString: STRING[80];
	DiagMessageIndex : UINT ; 
END_VAR

CASE eXMLReadState OF 
	LoadingFile :
		
		Busy:=TRUE;
		IF LoadFile THEN
		FileLoaded:= fbXml.LoadDocumentFromFile(
		sFile:= FileName,
		bExec:= LoadFile,
		);
		ELSE // file is loaded as fbXml has switched Loadfile to false so next step
			eXMLReadState := GettingIterator;
		END_IF

	
	GettingIterator : // this step navigates to the DiagMessages Node and initates the iterator
	IF NOT FileLoaded THEN 
		eXMLReadState := ErrorState;
	END_IF
		xmlDoc:= fbXml.GetDocumentNode();
		xmlEtherCatInfo := fbXml.ChildByName(xmlDoc, 'EtherCATInfo');
		xmlDescriptions := fbXml.ChildByName(xmlEtherCatInfo, 'Descriptions');
		xmlDevices := fbXml.ChildByName(xmlDescriptions, 'Devices');
		xmlDevice := fbXml.ChildByAttributeAndName(xmlDevices, 'Physics', 'YY', 'Device');
		xmlProfile := fbXml.ChildByName(xmlDevice, 'Profile');
		xmlDiagMessages := fbXml.ChildByName(xmlProfile, 'DiagMessages');
		xmlDiagmessageIterator:= fbXml.Begin(xmlDiagMessages);
		eXMLReadState := ParsingFile;
	
	ParsingFile : 
			FOR DiagMessageIndex:=0  TO NumToItetratePerCycle BY 1 DO // loop 0 to 25 
		IF NOT fbXml.IsEnd(xmlDiagmessageIterator) THEN// Still messages to Parse 
			xmlDiagMessage := fbXml.Node(xmlDiagmessageIterator); //  <DiagMessage> node
  			xmlDiagMessageIDNode :=  fbXml.ChildByName(xmlDiagMessage, 'TextId');// find the <TextID> in the level below 
			{analysis -26} // string possible truncated func gives 255 long string however only care about 6 chars so var is 8 char long
  			xmlDiagMessageIDText := fbXml.NodeText(xmlDiagMessageIDNode);// pull out the text 
			StringToUintError:= StringToUint(ErrorCodeString := xmlDiagMessageIDText ,ErrorCodeOut=> ErrorCode);
			xmlDiagMessageMessageTextNode :=  fbXml.ChildByName(xmlDiagMessage, 'MessageText');// find the <MessageText> 
	  		ErrorString := fbXml.NodeText(xmlDiagMessageMessageTextNode);// pull out the text, truncation of error string to 80 char warning
			 {analysis +26} 
			ErrorCodeStringArray[ErrorCode] := ErrorString;
			xmlDiagmessageIterator := fbXml.Next(xmlDiagmessageIterator);
		ELSE // out of messages
			eXMLReadState := Ready;	
		END_IF
		
		END_FOR
	
	Ready :
		ReadyFlag:= TRUE;
		Busy:= FALSE;
	ErrorState:
		Error:=TRUE;
		
	
	ELSE // in case a undefined Enum
		eXMLReadState := LoadingFile;
END_CASE

METHOD FB_init : BOOL
VAR_INPUT
	bInitRetains : BOOL; // if TRUE, the retain variables are initialized (warm start / cold start)
	bInCopyCode : BOOL;  // if TRUE, the instance afterwards gets moved into the copy code (online change)
	FileNameIn	: String[255];
END_VAR
FileName := FileNameIn;
END_METHOD

// returns true if a String is found for that error code
{attribute 'analysis' := '-23'} // complex return value for returning string 
METHOD Public GetErrorString : BOOL
VAR_INPUT
		ErrorCodeIn:UINT;
END_VAR
VAR_OUTPUT

		ErrorStringOut:STRING;
END_VAR
IF (ErrorCodeStringArray[ErrorCodeIn] = '')THEN
	GetErrorString := FALSE; 
ELSE
	GetErrorString := TRUE; 
END_IF
ErrorStringOut := ErrorCodeStringArray[ErrorCodeIn];
END_METHOD

// method used to take the strings in the ESI file in format '#xFFFF' and return a Uint
//bool returns true if it read two bytes false if not 
METHOD PRIVATE StringToUint :BOOL
VAR_INPUT
	ErrorCodeString :STRING[8];
END_VAR
VAR_OUTPUT 
	ErrorCodeOut :UINT;
END_VAR
VAR
	DataOutput : ARRAY[0..1] OF BYTE; // stores output of HEXSTR_TO_DATA function
	FormattedString :STRING[255];
	SpacedString : STRING[255];
	ErrorCodeTemp :UINT;
	BytesWrote:UDINT;
END_VAR
FormattedString := RIGHT (STR:= ErrorCodeString,SIZE:= 4); // removes'#x'
SpacedString := INSERT(STR1:= FormattedString,STR2:=' ', POS := 2); // inserts a space between bytes as its what HEXSTR_TO_DATA requires
{analysis -130} // Implicit expanding conversions from sizeof operator
BytesWrote:= HEXSTR_TO_DATA(sHex := SpacedString,pData:= ADR(DataOutput),cbData:= SIZEOF(DataOutput));// Function Wants 'AB CD'
ErrorCodeTemp := SHL(BYTE_TO_UINT(DataOutput[0]),8); // shift left so first byte is in correct place
ErrorCodeTemp := ErrorCodeTemp OR BYTE_TO_UINT(DataOutput[1]); // but second byte in place
IF NOT (BytesWrote=2) THEN 
	StringToUint:=FALSE;
ELSE
	ErrorCodeOut := ErrorCodeTemp;
	StringToUint:=TRUE;
END_IF
END_METHOD

END_FUNCTION_BLOCK

// POUs/FB_IDXResetError
FUNCTION_BLOCK FB_IDXResetError 
VAR_IN_OUT
	Execute			: BOOL;(*Function block execution is triggered by a rising edge at this input.*)
END_VAR

VAR_INPUT
	{attribute 'analysis' := '-35'} // is used in coe read dont understood why not picked up
	Axis			: AXIS_REF;
END_VAR
VAR
	AxisName :STRING;
	fbIDXErrorEventSender 	: FB_MotionEventSender;
	CoeMessageSent :BOOL;
	EventSent :BOOL;
	Busy :BOOL;
	stResetState : ST_MCState;
	
	fbCoEWrite		: FB_CoEWrite;
	Data       		: UINT := 16#0080;
    AdsErrId       	: UINT;
    CANopenErrId   	: UINT;
END_VAR
VAR CONSTANT
	NetId          	: T_AmsNetID:= '';(*netID of PC with NC*)
   	Index          	: WORD:= 16#6040;(*CoE object index*)
   	SubIndex       	: BYTE:=16#0;(*CoE sub index*)
   	Timeout        	: TIME := DEFAULT_ADS_TIMEOUT;(*States the time before the function is cancelled.*)
  	CompleteAccess 	: BOOL:= FALSE;(*Function block reads the complete object with all sub index*)
END_VAR

IF (stResetState.MCState = e_MCState.Done) THEN
	stResetState.MCState := e_MCState.Idle;
END_IF

IF __ISVALIDREF(Execute) THEN	
	fbCoEWrite(
    NetId          := NetId, 
    Index          := Index, 
    SubIndex       := SubIndex, 
    pSrcBuf        := ADR(Data), 
    BufLen         := USINT_TO_UDINT(SIZEOF(Data)), 
    Execute        := Execute, 
    Timeout        := Timeout, 
    CompleteAccess := CompleteAccess, 
    Axis := Axis,
	Busy => stResetState.Busy
); 
END_IF

IF (NOT Busy AND   __ISVALIDREF(Execute)) THEN
    stResetState.Error  := fbCoEWrite.Error;
    AdsErrId     		:= fbCoEWrite.AdsErrId;
    CANopenErrId 		:=fbCoEWrite.CANopenErrId;
    Execute      		:= FALSE;
	stResetState.MCState := e_MCState.Done;
END_IF

CoeMessageSent	:= fbIDXErrorEventSender.COEError(
	AxisName	:= AxisName,
	Error 		:= stResetState.Error,
	AdsErrId	:= AdsErrId,
	Description	:= 'ResettingAxis');
	
		
IF stResetState.Busy THEN
		stResetState.MCState := e_MCState.Busy;
END_IF

IF stResetState.Error THEN
	stResetState.MCState:= e_MCState.Error;
END_IF

EventSent:= fbIDXErrorEventSender.MotorReset(
	stAxisResetState:= stResetState,
	AxisName:= AxisName,
	ErrorCodeIn:= stResetState.ErrorID);

METHOD FB_init : BOOL
VAR_INPUT
	bInitRetains : BOOL; // if TRUE, the retain variables are initialized (warm start / cold start)
	bInCopyCode : BOOL;  // if TRUE, the instance afterwards gets moved into the copy code (online change)
	AxisNameIn :STRING;
END_VAR
AxisName := AxisNameIn;
END_METHOD

END_FUNCTION_BLOCK

// POUs/FB_Motion
FUNCTION_BLOCK FB_Motion
VAR_INPUT
END_VAR
VAR_OUTPUT
END_VAR
VAR
	Axis				: AXIS_REF;
	AxisName 			: STRING;
	fbMotionEventSender : FB_MotionEventSender;
	
	
	fbAxisPower			: MC_Power;
	stAxisPowerState 	: ST_MCState;
	
	fbAxisHalt 			: MC_Halt;
	stAxisHaltState 	: ST_MCState;
	
	fbAxisMove 			: MC_MoveAbsolute;
	stAxisMoveState 	: ST_MCState;
	
	fbAxisReset 		: MC_Reset;
	stAxisResetState 	:ST_MCState;
	
	fbAxisHome 			: MC_Home;
	stAxisHomeState 	: ST_MCState;
	
	NCErrorEventSent 	: BOOL;
END_VAR

Axis.ReadStatus();

NCErrorEventSent:= fbMotionEventSender.NCError(
	stAxisStatus := Axis.Status,
	AxisName := AxisName);

METHOD PUBLIC Enable : BOOL
VAR_INPUT
	Execute :BOOL;
END_VAR
VAR
	EventSent :bool;
END_VAR
Enable := FALSE;
fbAxisPower( // use in idx class
    Axis:= Axis,
    Enable:= Execute,
    Enable_Positive:= Execute,
    Enable_Negative:= Execute,
	BufferMode := MC_Aborting,
    Override:= 100.0,
	Status=>stAxisPowerState.Status,
	Error=>stAxisPowerState.Error,
	ErrorID => stAxisPowerState.ErrorID,
	Busy => stAxisPowerState.Busy
);

IF stAxisPowerState.Status THEN // axis is enabled
	stAxisPowerState.MCState := e_MCState.Active;
	Enable:= TRUE;
	
ELSIF stAxisPowerState.Busy THEN // fb is busy while enabling or axis is enabled
	stAxisPowerState.MCState := e_MCState.Busy;
	
ELSIF stAxisPowerState.Error THEN // in error state 
	stAxisPowerState.MCState := e_MCState.Error;
ELSE 
	stAxisPowerState.MCState := e_MCState.Idle;
END_IF


EventSent:= fbMotionEventSender.EnableMotor(
	stAxisPowerState:= stAxisPowerState,
	AxisName:= AxisName);
END_METHOD

METHOD Public Estop
VAR_INPUT
	Execute :bool;
END_VAR
fbAxisHalt(
	Axis:=Axis, 
	Execute:= Execute, 
	Deceleration:= , 
	Jerk:= , 
	BufferMode:=MC_Aborting ,  
	Done=> stAxisHaltState.Done, 
	Busy=>stAxisHaltState.Busy , 
	Active=>stAxisHaltState.Active , 
	CommandAborted=>stAxisHaltState.CommandAborted , 
	Error=>stAxisHaltState.Error , 
	ErrorID=> stAxisHaltState.ErrorID );
	
	

IF stAxisHaltState.Done THEN // axis been stopped 
		stAxisHaltState.MCState:= e_MCState.Done;
		
	ELSIF stAxisHaltState.Busy THEN 
		stAxisHaltState.MCState:= e_MCState.Busy;
		
	ELSIF stAxisHaltState.Error THEN	
		stAxisHaltState.MCState:= e_MCState.Error;
		
	ELSIF stAxisHaltState.CommandAborted THEN	
		stAxisHaltState.MCState:= e_MCState.CommandAborted;
		
	ELSE
		stAxisHaltState.MCState:= e_MCState.Idle;

	
END_IF
END_METHOD

METHOD FB_init : BOOL
VAR_INPUT
	bInitRetains : BOOL; // if TRUE, the retain variables are initialized (warm start / cold start)
	bInCopyCode : BOOL;  // if TRUE, the instance afterwards gets moved into the copy code (online change)
	AxisNameIn :string;
END_VAR
AxisName := AxisNameIn;
END_METHOD

METHOD PUBLIC GetAxisRef
VAR_IN_OUT
	AxisRefOut : AXIS_REF;
END_VAR
IF __ISVALIDREF(AxisRefOut) THEN
	AxisRefOut := Axis;	
END_IF
END_METHOD

METHOD PUBLIC GetCurrentPosition
VAR_OUTPUT
	PositionOut :LREAL;
END_VAR
PositionOut:= Axis.NcToPlc.ActPos;
END_METHOD

METHOD public GetStatus 
VAR_IN_OUT
	AxisOut :ST_AxisStatus;
END_VAR
IF __ISVALIDREF(AxisOut) THEN
	AxisOut := Axis.Status;
END_IF
END_METHOD

METHOD PUBLIC Home : BOOL
VAR_IN_OUT
	Execute :BOOL;
END_VAR

VAR_INPUT
		HomePositionIn :LREAL;
END_VAR
VAR
	HomeEventSent		: BOOL;
END_VAR
IF __ISVALIDREF(Execute) THEN
	
	fbAxisHome(
		Axis:=Axis,
		Execute:=Execute,
		Position:=HomePositionIn,
		HomingMode:=MC_DefaultHoming,
		Busy=>stAxisHomeState.Busy,
		Done=>stAxisHomeState.Done,
		Error=> stAxisHomeState.Error,
		ErrorID=> stAxisHomeState.ErrorID);

	
	IF stAxisHomeState.Done THEN // axis been Homed 
		stAxisHomeState.MCState:= e_MCState.Done;
		
		ELSIF stAxisHomeState.Busy THEN // 
			stAxisHomeState.MCState:= e_MCState.Busy;
		
		ELSIF stAxisHomeState.Error THEN	
			stAxisHomeState.MCState:= e_MCState.Error;
		
		ELSIF stAxisHomeState.CommandAborted THEN	
			stAxisHomeState.MCState:= e_MCState.CommandAborted;
		
		ELSE
			stAxisHomeState.MCState:= e_MCState.Idle;

	END_IF

	IF stAxisHomeState.Busy THEN
		Execute := FALSE;
	END_IF
END_IF

 Home:= stAxisHomeState.Busy;
 
HomeEventSent:= fbMotionEventSender.Homing(
	stAxisHomeState:= stAxisHomeState,
	AxisName:= AxisName
	);
END_METHOD

METHOD PUBLIC MoveTo : BOOL
VAR_INPUT
	TargetPositionIn : LREAL;
	VelocityIn : LREAL;
END_VAR

VAR_IN_OUT
		Execute :BOOL;
END_VAR
VAR_OUTPUT
	eStateOut : e_MCState;
END_VAR
VAR
	EventSent	: bool;
END_VAR

IF  __ISVALIDREF(Execute) THEN
	fbAxisMove(
		Axis:= Axis, 
		Execute:= Execute, 
		Position:= TargetPositionIn, 
		Velocity:= VelocityIn, 
		BufferMode:= MC_BufferMode.MC_BlendingNext , 
		Done=>stAxisMoveState.Done , 
		Busy=> stAxisMoveState.Busy, 
		Active=> stAxisMoveState.Active, 
		CommandAborted=> stAxisMoveState.CommandAborted, 
		Error=>stAxisMoveState.Error , 
		ErrorID=> stAxisMoveState.ErrorID);
	
	IF stAxisMoveState.Active THEN // axis In Motion
		stAxisMoveState.MCState:= e_MCState.Active;
		
		ELSIF stAxisMoveState.Busy THEN // fb busy
			stAxisMoveState.MCState:= e_MCState.Busy;
		
		ELSIF stAxisMoveState.Error THEN	
			stAxisMoveState.MCState:= e_MCState.Error;
		
		ELSIF stAxisMoveState.CommandAborted THEN	
			stAxisMoveState.MCState:= e_MCState.CommandAborted;
		
		ELSIF stAxisMoveState.Done THEN
			stAxisMoveState.MCState := e_MCState.Done;
		
		ELSE
			stAxisMoveState.MCState:= e_MCState.Idle;

	END_IF

	eStateOut:= stAxisMoveState.MCState;

	IF stAxisMoveState.Busy THEN
		Execute := FALSE;
	END_IF
END_IF

EventSent:= fbMotionEventSender.MoveTo(
	stAxisMoveState:= stAxisMoveState,
	AxisName:= AxisName,
	TargetPositionIn:= TargetPositionIn,
	VelocityIn:= VelocityIn);
END_METHOD

METHOD PUBLIC Reset : BOOL
VAR_IN_OUT
	Execute:BOOL;
END_VAR

VAR
ResetEventSent :bool;
END_VAR
Reset := FALSE;
IF  __ISVALIDREF(Execute) THEN
	fbAxisReset(
		Axis:= Axis, 
		Execute:= Execute, 
		Done=> stAxisResetState.Done, 
		Busy=> stAxisResetState.Busy, 
		Error=>stAxisResetState.Error , 
		ErrorID=>stAxisResetState.ErrorID);

	
	IF stAxisResetState.Done THEN
		stAxisResetState.MCState := e_MCState.Done;
		Reset := TRUE;
		Execute:= FALSE;
		
	ELSIF stAxisResetState.Busy THEN
		stAxisResetState.MCState := e_MCState.Busy;
	END_IF

	IF stAxisResetState.Error THEN
		stAxisResetState.MCState:= e_MCState.Error;
	END_IF

	IF NOT (stAxisResetState.Error OR stAxisResetState.Busy OR stAxisResetState.Done) THEN
		stAxisResetState.MCState:= e_MCState.Idle;
	END_IF

END_IF

ResetEventSent:= fbMotionEventSender.NCReset(
	stAxisResetState:= stAxisResetState,
	AxisName:= AxisName,
	ErrorCodeIn:= stAxisResetState.ErrorID);
END_METHOD

END_FUNCTION_BLOCK

// POUs/FB_MotorBrake
// fb to manage brake events will be sent for error aswell as a error boolean 
// to be run every cycle 
FUNCTION_BLOCK PUBLIC FB_MotorBrake
VAR_INPUT
END_VAR
VAR_OUTPUT
	Status :e_IDXBrakeState;
END_VAR
VAR
	BrakeOutput				:BOOL; // desired state
	BrakeValveOutput 		:BOOL; // mapped to send to 3/2 valve
	EngagementSensor		:BOOL; // 1 is brake engaged 0 is disengaged so movement is possible
	SafetySystemOverride	:BOOL; // 1 means safety system has brake applied 
	MaxBrakeActivateTime	:TIME; // max time in ms between no signal and activing 
	MaxBrakeDeactivateTime	:TIME; // max time in ms between signal and releasing
	EngageTimer 			:TON;
	EngageTimerIn 			:BOOL;
	DisengageTimer 			:TON;
	_Error 					:BOOL;
	EngageTimerError 		:BOOL;
	DisengageTimerError		:BOOL;
	AirPressureError		:BOOL;
	AirPressure 			:REAL; // in bar 
	MinAirPressure			:REAL;
	AxisName 				:STRING;
	BrakeStatus 			:e_IDXBrakeState:= e_IDXBrakeState.Unknown;
	DisengagementTimerIn	:BOOL;
	ErrorAck				:BOOL:= FALSE;
END_VAR

EngageTimer(IN:=EngageTimerIn);
DisengageTimer(IN:= DisengagementTimerIn);

// check for  safety system activation
IF SafetySystemOverride AND NOT ((BrakeStatus=  e_IDXBrakeState.SafetyOverriden) OR (BrakeStatus=  e_IDXBrakeState.SafetyActivating) ) THEN
	IF EngagementSensor THEN
		BrakeStatus := e_IDXBrakeState.SafetyOverriden;
	ELSE
		BrakeStatus := e_IDXBrakeState.SafetyActivating;
	END_IF
END_IF

IF EngageTimerError OR DisengageTimerError THEN
	BrakeStatus := e_IDXBrakeState.Error;
END_IF

// check for airpressure Fault
IF AirPressure<MinAirPressure THEN
	AirPressureError := TRUE;
ELSE
	AirPressureError := FALSE;
END_IF

IF AirPressureError AND NOT  (BrakeStatus = e_IDXBrakeState.Error) THEN 
	BrakeStatus := e_IDXBrakeState.Unpowered;
END_IF

CASE(BrakeStatus) OF 
e_IDXBrakeState.Unpowered:// no air
	BrakeOutput := TRUE;
	BrakeValveOutput:= FALSE; // so doesnt rapidly disengage on air restoration
	IF AirPressure>MinAirPressure THEN
		BrakeStatus:= e_IDXBrakeState.Engaged;
	END_IF

e_IDXBrakeState.Engaged:// brake engaged check for brake output switching and move to disengaging
DisengagementTimerIn:= FALSE;
EngageTimerIn:= FALSE;
IF NOT BrakeOutput THEN
	BrakeValveOutput :=TRUE;
	BrakeStatus := e_IDXBrakeState.Disengaging;
END_IF

e_IDXBrakeState.Disengaging: // brake disengaging timer to check for errors 
	DisengagementTimerIn:= TRUE;
	IF DisengageTimer.Q THEN
		DisengageTimerError:= TRUE;
	END_IF
	IF NOT EngagementSensor THEN
		BrakeStatus:= e_IDXBrakeState.Disengaged;
	END_IF

e_IDXBrakeState.Disengaged: // brake disengaged check for output switching move to engaging
	DisengagementTimerIn:= FALSE;
	EngageTimerIn:= FALSE;
	IF BrakeOutput THEN
		BrakeValveOutput :=FALSE;
		BrakeStatus := e_IDXBrakeState.Engaging;
	END_IF
	
	
	
e_IDXBrakeState.Engaging: 
	EngageTimerIn:= TRUE;
	IF EngageTimer.Q THEN
		EngageTimerError:= TRUE;
	END_IF
	IF EngagementSensor THEN
		BrakeStatus:= e_IDXBrakeState.Engaged;
	END_IF
 

e_IDXBrakeState.SafetyOverriden: // brake engaged by safety system check if non overridden any more and move to engaged also reset timers 
	DisengagementTimerIn:= FALSE;
	EngageTimerIn:= FALSE;
	BrakeOutput := TRUE;
	BrakeValveOutput:= FALSE; // so doesnt rapidly disengage on safety reset
	IF NOT SafetySystemOverride THEN
		BrakeStatus:= e_IDXBrakeState.Engaged;
	END_IF
	

e_IDXBrakeState.SafetyActivating: // brake engaging by safety system check for system over ride tthrow in here then check when its engaged resettimers 
EngageTimerIn:= TRUE;
	IF EngageTimer.Q THEN
		EngageTimerError:= TRUE;
	END_IF
	IF EngagementSensor THEN
		BrakeStatus:= e_IDXBrakeState.SafetyOverriden;
	END_IF

e_IDXBrakeState.Unknown: // try to figure out status from inputs reset timers 
	IF AirPressure<MinAirPressure THEN
		BrakeStatus:= e_IDXBrakeState.Unpowered;
	ELSE // got air pressure 
		IF SafetySystemOverride THEN
			IF EngagementSensor THEN
				BrakeStatus := e_IDXBrakeState.SafetyOverriden;
			ELSE
				BrakeStatus := e_IDXBrakeState.SafetyActivating;
			END_IF
		ELSE //not safety overriden
			IF EngagementSensor THEN
				BrakeStatus := e_IDXBrakeState.Engaged;
			ELSE
				BrakeStatus := e_IDXBrakeState.Disengaged;
			END_IF
		END_IF
	END_IF

	e_IDXBrakeState.Error: //overran timing
	BrakeOutput := TRUE;
	BrakeValveOutput:= FALSE;
	DisengagementTimerIn:= FALSE;
	EngageTimerIn:= FALSE;
	IF ErrorAck THEN
		DisengageTimerError:= FALSE;
		EngageTimerError := FALSE;
		BrakeStatus := e_IDXBrakeState.Unknown;
		ErrorAck := FALSE;
	END_IF
	
	

ELSE
	BrakeStatus := e_IDXBrakeState.Unknown;

END_CASE

Status:= BrakeStatus;
// error events including resetting the 
_error := EngageTimerError OR DisengageTimerError OR AirPressureError;
 // error if overridden

// used to active and deactivate brake
METHOD PUBLIC Brake : BOOL // returns a boolean once brake is activated
VAR_IN_OUT
	Engage : BOOL;
END_VAR
VAR_OUTPUT
	Error :BOOL; // true if brake not activating 
END_VAR

// if error is triggered then change the enable signal to brakes current state 
IF _error THEN// 
	Engage := TRUE; // in error put brake on 
END_IF
BrakeOutput:= Engage;// transfer desired state
Brake:=EngagementSensor;// output bool of funct
Error := _Error;
END_METHOD

// used to check current brake status 
METHOD PUBLIC BrakeStatus : BOOL
VAR_INPUT
END_VAR
BrakeStatus := EngagementSensor;
END_METHOD

// function deals with the brake and enabling the motor in one function 
METHOD EnableMotor : BOOL
VAR_INPUT
	Execute :BOOL;
	fbMotionInstance :REFERENCE TO fb_motion;
	Error :bool;
END_VAR
END_METHOD

METHOD FB_init : BOOL
VAR_INPUT
	bInitRetains : BOOL; // if TRUE, the retain variables are initialized (warm start / cold start)
	bInCopyCode : BOOL;  // if TRUE, the instance afterwards gets moved into the copy code (online change)
	MaxBrakeActivateTimein:TIME;//  max time in ms between no signal and activing 
	MaxBrakeDeactivateTimein:TIME;//  max time in ms between signal and releasing
	MinAirPressureIn:REAL;
END_VAR
EngageTimer.PT:= MaxBrakeActivateTimein;
DisengageTimer.PT := MaxBrakeActivateTimein;
MinAirPressure:= MinAirPressureIn;
//BrakeActiveTimer(PT:= MaxBrakeActivateTimein);
//BrakeDeactiveTimer(PT:= MaxBrakeActivateTimein);
END_METHOD

METHOD UnitTestInputs 
VAR_INPUT
	EngagementSensorIn:BOOL;
	AirPressureIn :REAL;
	SafetySystemOverrideIn:BOOL;
END_VAR
EngagementSensor:= EngagementSensorIn;
AirPressure:= AirPressureIn;
SafetySystemOverride:= SafetySystemOverrideIn;
END_METHOD

END_FUNCTION_BLOCK

// POUs/MAIN
{attribute 'analysis' := '-33,-2'}
PROGRAM MAIN
VAR

END_VAR

END_PROGRAM
